Staubli VAL3: oEmergencyOut.pgx

public program oEmergencyOut(num nChoice (dimensions=1))
// oEmergencyOut
begin
  dioSet(oEmergencyOut,nChoice)
end
